// TIA Portal V17 export
// export: Created 2023-04-03T06:31:43.9665748Z, ExportSetting WithDefaults, DisplayName Totally Integrated Automation Portal, DisplayVersion V17 Update 4, DisplayName TIA Portal Openness, DisplayVersion V17 Update 4, DisplayName TIA Portal Version Control Interface, DisplayVersion V17, DisplayName STEP 7 Professional, DisplayVersion V17 Update 4, DisplayName STEP 7 Safety, DisplayVersion V17, DisplayName WinCC Professional, DisplayVersion V17 Update 4
TYPE "BR"
// stored: IsFailsafeCompliant false
   STRUCT
      iAssetSt : Int;
      rVcellAvg : Real;
      iTcellAvg : Int;
      rIdc : Real;
      rVcellMax : Real;
      iVmodMaxPos : Int;
      iTcellMax : Int;
      iTmodMaxPos : Int;
      rVcellMin : Real;
      iVmodMinPos : Int;
      iTcellMin : Int;
      iTmodMinPos : Int;
      rSOC : Real;
      rSOH : Real;
      rVdc : Real;
      iTrackIn : Int;
      iTrackOut : Int;
      iTamb : Int;
      iTempSet : Int;
   END_STRUCT;
END_TYPE
